FUNCTION_BLOCK XtsMover IMPLEMENTS IMover
VAR_INPUT
END_VAR
VAR_OUTPUT
END_VAR
VAR
	axesEnable		: MC_Power;
	axesReset		: AxesReset(_axis);
	axesMoveTo 		: MoveMoverToPositionZoned(_axis) := (Gap := 213.0);
	axesHalt 		: HaltMover(_axis);
	axesReadError : Tc2_MC2.MC_ReadAxisError;
	_axis 			: AXIS_REF;
	_identInGroup : INT;
	_trackLength : REAL;
	_targetPos : LREAL;
	_MoverErrorId : DWORD;
	_arrZones : ARRAY[1..4] OF DINT;
	_arrVelocities : ARRAY[1..4] OF mc_LREAL;
END_VAR

axesMoveTo(arrPositions := _arrZones, arrVelos := _arrVelocities);
axesHalt();
axesReset();
_axis.ReadStatus();
axesEnable(Axis := _axis);
axesReadError(Axis := _axis, Enable := TRUE, AxisErrorID => _MoverErrorId);

PROPERTY PUBLIC Acceleration : mc_lreal
GET
Acceleration := axesMoveTo.Acceleration;
END_GET
SET
axesMoveTo.Acceleration := Acceleration;
END_SET
END_PROPERTY

PROPERTY PUBLIC AxisRef : reference to AXIS_REF
GET
AxisRef REF= THIS^._axis;
END_GET
END_PROPERTY

PROPERTY PUBLIC Deceleration : mc_lreal
GET
Deceleration := axesMoveTo.Deceleration;
END_GET
SET
axesMoveTo.Deceleration := Deceleration;
END_SET
END_PROPERTY

METHOD PUBLIC DisableAxis : BOOL
VAR_INPUT
END_VAR
axesEnable.Enable := false;
END_METHOD

METHOD PUBLIC EnableAxis : BOOL
VAR_INPUT
END_VAR
axesEnable.Enable := axesEnable.Enable_Negative := axesEnable.Enable_Positive := TRUE;
axesEnable.Override := 100;
END_METHOD

PROPERTY PUBLIC Gap : mc_lreal
GET
Gap := axesMoveTo.Gap;
END_GET
SET
axesMoveTo.Gap := Gap;
END_SET
END_PROPERTY

METHOD PUBLIC HaltAxis : BOOL
VAR_INPUT
END_VAR
IF NOT axesHalt.Busy THEN
	axesHalt.Execute();
	HaltAxis := TRUE;
END_IF
END_METHOD

METHOD hasError : BOOL
VAR_INPUT
END_VAR
hasError := _axis.Status.Error;
END_METHOD

PROPERTY PUBLIC IdentInGroup : int
GET
IdentInGroup := _identInGroup;
END_GET
SET
_identInGroup := IdentInGroup;
END_SET
END_PROPERTY

METHOD isAtPosition : BOOL
VAR_INPUT
	position : MC_LREAL;
END_VAR
IF position > 1 THEN
	IF _axis.NcToPlc.ModuloActPos < position + 1 AND _axis.NcToPlc.ModuloActPos > position - 1 THEN
		isAtPosition := TRUE;
	END_IF  
ELSE
	IF _axis.NcToPlc.ModuloActPos < position + 1 AND _axis.NcToPlc.ModuloActPos > 0.0  
		OR _axis.NcToPlc.ModuloActPos < _trackLength AND _axis.NcToPlc.ModuloActPos > _trackLength - 1 THEN
		isAtPosition := TRUE;
	END_IF
END_IF
END_METHOD

METHOD PUBLIC isDetected : BOOL
VAR_INPUT
END_VAR
IF _axis.NcToPlc.AxisId = 0 THEN
	RETURN;
END_IF
isDetected := true;
END_METHOD

METHOD isEnabled : BOOL
VAR_INPUT
END_VAR
isEnabled := not _axis.Status.Disabled;
END_METHOD

PROPERTY PUBLIC Jerk : mc_lreal
GET
Jerk := axesMoveTo.Jerk;
END_GET
SET
axesMoveTo.Jerk := Jerk;
END_SET
END_PROPERTY

METHOD PRIVATE ModuloToAbs : mc_lreal
VAR_INPUT
	moduloPositionDemand: MC_LREAL;
	_backwardsAllowed : BOOL;
END_VAR
//---------code to set actual position from modulo command----------------------
IF NOT _backwardsAllowed THEN
	//--------if you want to go forward-------------------------------------------------------------
	//---------if SetPos is greater than current actual then move to that position--------------------
	//---------else current position is greater, increase moduloturn count by 1 before set---------------
	IF moduloPositionDemand > _axis.NcToPlc.ModuloActPos THEN
		ModuloToAbs := (_Axis.NcToPlc.ModuloActTurns*_trackLength) + moduloPositionDemand;
	ELSE
		ModuloToAbs := ((_Axis.NcToPlc.ModuloActTurns + 1)*_trackLength) + moduloPositionDemand;
	END_IF
ELSE
	//--------if you want to go backwards--------------------------------
	//--------if setPos is less than current actual then move to that position---------------------
	//---------else current position is less, decrease moduloturn count by 1 before set------------
	IF moduloPositionDemand < _axis.NcToPlc.ModuloActPos THEN
		ModuloToAbs := (_Axis.NcToPlc.ModuloActTurns*_trackLength) + moduloPositionDemand;
	ELSE
		ModuloToAbs := ((_Axis.NcToPlc.ModuloActTurns-1)*_trackLength) + moduloPositionDemand;
		//ModuloToAbsolute := ((_Axis.NcToPlc.ModuloActTurns - 1)*GVLAxesRefs.iXTSTrackLength) + moduloPositionDemand;
	END_IF
END_IF
END_METHOD

PROPERTY MoverErrorId : dword
GET
MoverErrorId := _MoverErrorId;
END_GET
SET
_MoverErrorId := MoverErrorId;
END_SET
END_PROPERTY

METHOD PUBLIC MoveTo : BOOL
VAR_INPUT
	Position : MC_LREAL;
	Velocity : MC_LREAL;
	BackwardMove : BOOL;
END_VAR
IF NOT isAtPosition(position := Position) THEN
	IF NOT axesMoveTo.Busy THEN
		axesMoveTo.MoveTo(Position := ModuloToAbs(Position, BackwardMove), Velocity := Velocity);
		MoveTo := TRUE;
		_targetPos := Position;
	END_IF
END_IF
END_METHOD

METHOD PUBLIC ResetAxis : BOOL
VAR_INPUT
END_VAR
VAR
END_VAR
axesReset.Execute();
axesMoveTo.Abort();
axesHalt.Abort();
END_METHOD

PROPERTY PUBLIC TrackLength : real
GET
TrackLength := _trackLength;
END_GET
SET
_trackLength := TrackLength;
END_SET
END_PROPERTY

PROPERTY Zones : array[1..4] of dint
GET
Zones := _arrZones;
END_GET
SET
_arrZones := Zones;
END_SET
END_PROPERTY

PROPERTY ZoneVelocities : array[1..4] of mc_lreal
GET
ZoneVelocities := _arrVelocities;
END_GET
SET
_arrVelocities := ZoneVelocities;
END_SET
END_PROPERTY

END_FUNCTION_BLOCK

(* stored: Version 1.1.0.1, ProductVersion 3.1.4024.6
   POU XtsMover: Id {203ccb09-708b-4f54-b5b6-0f120d67335b}, SpecialFunc None
   Folder Methods: Id {bc3bf09c-c7d7-4024-96a7-671bf690c24c}
   Folder Properties: Id {62e911ec-7686-46c6-839c-cb7436ba3335}
   Property Acceleration: Id {4e5a89d0-785e-4c3f-b801-4d01ed56f986}
   Get Get: Id {a063cc41-5faf-4d0c-b1e5-75c373e5685c}
   Set Set: Id {16a025f3-6684-4a8e-94ea-54a03cd581c6}
   Property AxisRef: Id {9b58505a-2998-4f2c-b04d-fff116217974}
   Get Get: Id {d9e4a655-8a01-4876-94ff-b6745986fc39}
   Property Deceleration: Id {2da8c65a-ea43-4ee7-b0b8-dd1d445fda83}
   Get Get: Id {5d613a9f-9c38-4460-bdcb-fbb36f5d571e}
   Set Set: Id {0f6bce91-7c89-451e-a5b3-554db1d234e8}
   Method DisableAxis: Id {d1142462-06a0-4086-877d-bf769eaaeb65}
   Method EnableAxis: Id {98c94290-90b2-404d-90db-c6c3a781b1ed}
   Property Gap: Id {30f92ef9-8876-4a21-9385-112c82c14c10}
   Get Get: Id {8bf691ac-11b3-468f-bd60-47c1a98bb6f6}
   Set Set: Id {ed2230ca-9b27-40f6-a0a6-89da0bd85186}
   Method HaltAxis: Id {46252ae4-f527-4552-9d65-581a4a2179e1}
   Method hasError: Id {6a2c6507-492c-4ada-a24d-ccb9597917f5}
   Property IdentInGroup: Id {cec3e36d-fd9f-4a09-8f93-73f82a502874}
   Get Get: Id {18684a3b-73b2-42c3-bf7c-d412f63c526e}
   Set Set: Id {1dceadc0-b86b-4bcf-a0f9-102e0cec8ef8}
   Method isAtPosition: Id {a096a07e-dab0-4256-a3b3-e56e1c2d96f7}
   Method isDetected: Id {93d0b88b-b65a-4881-bf5d-1938b7f668bf}
   Method isEnabled: Id {349e6766-2db0-4f6c-8069-dc9579f83c27}
   Property Jerk: Id {8dbc2563-ca56-48eb-bdb2-972740f27e21}
   Get Get: Id {a6c375d2-6153-4e85-a1a3-18b06e9113be}
   Set Set: Id {eacd414b-102d-4797-8934-580093cdc6ca}
   Method ModuloToAbs: Id {b920ad30-7e5c-4a74-b883-c04a36c8b0f9}
   Property MoverErrorId: Id {fa6a010c-2b2c-487f-8a34-7485c92b0387}
   Get Get: Id {fe3cb620-7c11-4f42-a3c1-8fdaebb297ac}
   Set Set: Id {b27ba25f-cedc-4b1b-a21c-51101e941d22}
   Method MoveTo: Id {1a78ba9e-748f-4851-bb07-1880a777b968}
   Method ResetAxis: Id {627dcfae-96a6-483b-aeaf-b2bb92851eed}
   Property TrackLength: Id {d175efd0-8db6-42ab-b883-df9200333ebe}
   Get Get: Id {1670d4fa-76f9-4278-871b-e1f420319691}
   Set Set: Id {14b136df-3930-4f12-921f-2ee26b4b33d6}
   Property Zones: Id {1e1c9dad-3c7f-4e75-bceb-b4591f5bd64f}
   Get Get: Id {8c2c8a28-5b87-4fa4-8e82-43aacf62a5e3}
   Set Set: Id {67c21546-1db6-45a1-ad68-905fc1bc605c}
   Property ZoneVelocities: Id {d287b0eb-d15a-4f54-b384-d18650a4ca53}
   Get Get: Id {8d1af704-520b-4e30-af4c-83cbc62b0b7b}
   Set Set: Id {2cd34126-a7ab-43aa-b55b-a90d4ab8e7ec} *)
